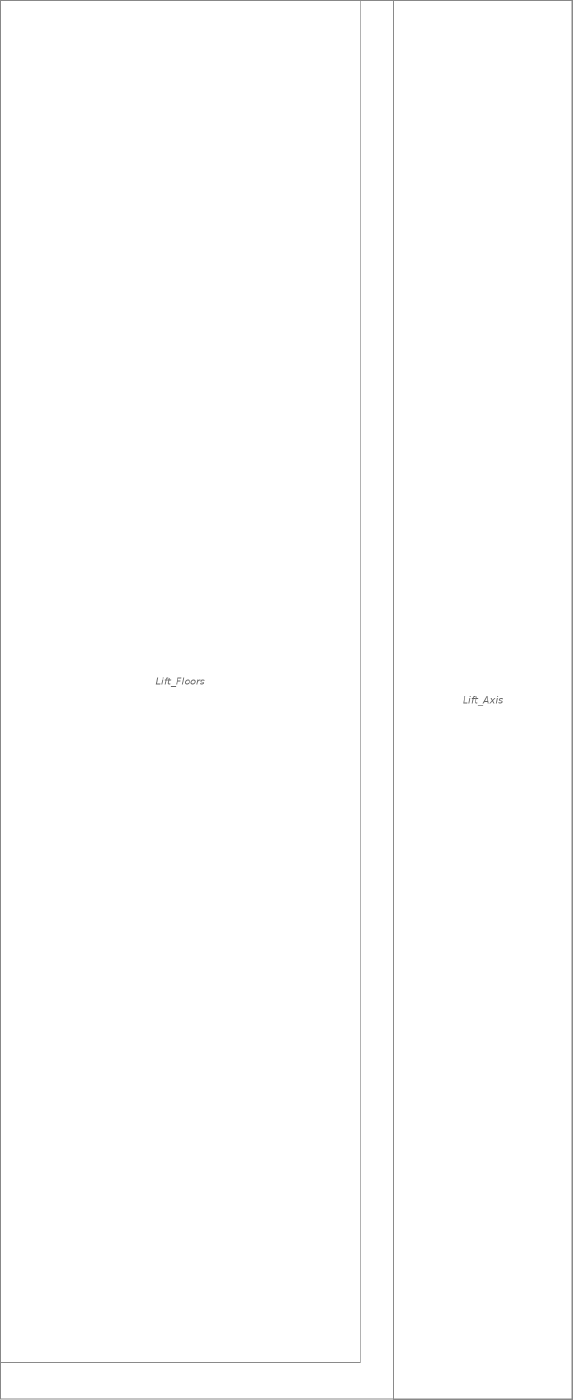
VISUALIZATION Lift  // 598x1461
VAR_IN_OUT
	Position : REAL;
	RefSensor : BOOL;
	Color : DWORD;
	Door_1_Position	: REAL;
	Door_1_M_Open	: BOOL;
	Door_1_M_Close	: BOOL;
	Door_2_Position	: REAL;
	
	Door_2_M_Open	: BOOL;
	Door_2_M_Close	: BOOL;
	Door_3_Position	: REAL;
	
	Door_3_M_Open	: BOOL;
	Door_3_M_Close	: BOOL;
	Door_4_Position	: REAL;
	
	Door_4_M_Open	: BOOL;
	Door_4_M_Close	: BOOL;
	Door_5_Position	: REAL;
	
	Door_5_M_Open	: BOOL;
	Door_5_M_Close	: BOOL;
	Door_6_Position	: REAL;
	
	Door_6_M_Open	: BOOL;
	Door_6_M_Close	: BOOL;
	LED_Up_1 		: BOOL;
	LED_Down_1 		: BOOL;
	FloorNumber_1 	: INT;
	BtnLed_1 		: ARRAY[1..6] OF BOOL;;
	Btn_1			: ARRAY[1..6] OF BOOL;
	LB_1 			: BOOL;
	LED_DoorOpen_1 	: BOOL;
	LED_DoorClosed_1: BOOL;

	LED_Up_2 		: BOOL;
	LED_Down_2 		: BOOL;
	FloorNumber_2 	: INT;
	BtnLed_2 		: ARRAY[1..6] OF BOOL;;
	Btn_2			: ARRAY[1..6] OF BOOL;
	LB_2 			: BOOL;
	LED_DoorOpen_2 	: BOOL;
	LED_DoorClosed_2: BOOL;


	LED_Up_3 		: BOOL;
	LED_Down_3 		: BOOL;
	FloorNumber_3 	: INT;
	BtnLed_3 		: ARRAY[1..6] OF BOOL;;
	Btn_3			: ARRAY[1..6] OF BOOL;
	LB_3 			: BOOL;
	LED_DoorOpen_3 	: BOOL;
	LED_DoorClosed_3: BOOL;

	LED_Up_4 		: BOOL;
	LED_Down_4 		: BOOL;
	FloorNumber_4 	: INT;
	BtnLed_4 		: ARRAY[1..6] OF BOOL;;
	Btn_4			: ARRAY[1..6] OF BOOL;
	LB_4 			: BOOL;
	LED_DoorOpen_4 	: BOOL;
	LED_DoorClosed_4: BOOL;

	LED_Up_5 		: BOOL;
	LED_Down_5 		: BOOL;
	FloorNumber_5 	: INT;
	BtnLed_5 		: ARRAY[1..6] OF BOOL;;
	Btn_5			: ARRAY[1..6] OF BOOL;
	LB_5 			: BOOL;
	LED_DoorOpen_5 	: BOOL;
	LED_DoorClosed_5: BOOL;

	LED_Up_6 		: BOOL;
	LED_Down_6 		: BOOL;
	FloorNumber_6 	: INT;
	BtnLed_6 		: ARRAY[1..6] OF BOOL;;
	Btn_6			: ARRAY[1..6] OF BOOL;
	LB_6 			: BOOL;
	LED_DoorOpen_6 	: BOOL;
	LED_DoorClosed_6: BOOL;

END_VAR
    Frame (410,0 188x1461)
        shows Lift_Axis(Position := Visu_L1.Position_LIFT, RefSensor := RefSensor)
    Frame (0,0 376x1422)
        shows Lift_Floors(Color := Color, Door_1_Position := Door_1_Position, Door_1_M_Open := Door_1_M_Open, Door_1_M_Close := Door_1_M_Close, Door_2_Position := Door_2_Position, Door_2_M_Open := Door_2_M_Open, Door_2_M_Close := Door_2_M_Close, Door_3_Position := Door_3_Position, Door_3_M_Open := Door_3_M_Open, Door_3_M_Close := Door_3_M_Close, Door_4_Position := Door_4_Position, Door_4_M_Open := Door_4_M_Open, Door_4_M_Close := Door_4_M_Close, Door_5_Position := Door_5_Position, Door_5_M_Open := Door_5_M_Open, Door_5_M_Close := Door_5_M_Close, Door_6_Position := Door_6_Position, Door_6_M_Open := Door_6_M_Open, Door_6_M_Close := Door_6_M_Close, LED_Up_1 := LED_Up_1, LED_Down_1 := LED_Down_1, FloorNumber_1 := FloorNumber_1, BtnLed_1 := BtnLed_1, Btn_1 := Btn_1, LB_1 := LB_1, LED_DoorOpen_1 := LED_DoorOpen_1, LED_DoorClosed_1 := LED_DoorClosed_1, LED_Up_2 := LED_Up_2, LED_Down_2 := LED_Down_2, FloorNumber_2 := FloorNumber_2, BtnLed_2 := BtnLed_2, Btn_2 := Btn_2, LB_2 := LB_2, LED_DoorOpen_2 := LED_DoorOpen_2, LED_DoorClosed_2 := LED_DoorClosed_2, LED_Up_3 := LED_Up_3, LED_Down_3 := LED_Down_3, FloorNumber_3 := FloorNumber_3, BtnLed_3 := BtnLed_3, Btn_3 := Btn_3, LB_3 := LB_3, LED_DoorOpen_3 := LED_DoorOpen_3, LED_DoorClosed_3 := LED_DoorClosed_3, LED_Up_4 := LED_Up_4, LED_Down_4 := LED_Down_4, FloorNumber_4 := FloorNumber_4, BtnLed_4 := BtnLed_4, Btn_4 := Btn_4, LB_4 := LB_4, LED_DoorOpen_4 := LED_DoorOpen_4, LED_DoorClosed_4 := LED_DoorClosed_4, LED_Up_5 := LED_Up_5, LED_Down_5 := LED_Down_5, FloorNumber_5 := FloorNumber_5, BtnLed_5 := BtnLed_5, Btn_5 := Btn_5, LB_5 := LB_5, LED_DoorOpen_5 := LED_DoorOpen_5, LED_DoorClosed_5 := LED_DoorClosed_5, LED_Up_6 := LED_Up_6, LED_Down_6 := LED_Down_6, FloorNumber_6 := FloorNumber_6, BtnLed_6 := BtnLed_6, Btn_6 := Btn_6, LB_6 := LB_6, LED_DoorOpen_6 := LED_DoorOpen_6, LED_DoorClosed_6 := LED_DoorClosed_6)
END_VISUALIZATION

(* stored: Version 1.1.0.1
   Visu Lift: Id {ab8a0c48-1bc1-404d-a4b9-4ca585106429} *)
